TYPE ST_SafeEL1918Status :
STRUCT
	State AT%I* :USINT;
	Diag AT%I* :USINT;
	Status :st_SafetyStatus;
	Inputs AT%I* :st_EL1918Inputs;
END_STRUCT
END_TYPE

(* stored: Version 1.1.0.1, ProductVersion 3.1.4024.12
   DUT ST_SafeEL1918Status: Id {d1faea2f-8be0-4661-9169-14610738a684} *)
